TYPE ST_MotorStatus :
STRUCT
    Running : BOOL;
END_STRUCT
END_TYPE

(* stored: Version 1.1.0.1, ProductVersion 3.1.4024.12
   DUT ST_MotorStatus: Id {22a17f96-5698-4da9-9059-29ca16dd29ce} *)
